(*
version 1.1	20. apr. 2008
programmer 	hugo
tested by	oscat

this function calculates the phase angle (argument) of a complex number

*)
FUNCTION CARG : REAL
VAR_INPUT
	X : complex;
END_VAR

CARG := ATAN2(X.im, X.re);



(* revision history
hm	21. feb. 2008	rev 1.0
	original version

hm	20. apr. 2008	rev 1.1
	use ATAN2 instead of ATAN
*)

END_FUNCTION

(* stored: Version 1.1.0.1
   POU CARG: Id {6a924c3c-d7ef-48cc-b786-e7eb257a799b}, SpecialFunc None *)
